// TIA Portal project "test3Servo" (V15.1)

(* hardware
DEVICE "S7-1200 station_1"  S7-1200 Station
   slot 0: "Rack_0"  S7-1200 Rack  Rack  V1.0
   slot 1: "PLC_1"  CPU 1217C DC/DC/DC  6ES7 217-1AG40-0XB0  V4.1
*)

// ===== PLC "PLC_1"  CPU 1217C DC/DC/DC =====

VAR_GLOBAL   // PLC tag table "Default tag table"
   "B1_Pulse" AT %Q0.0 : Bool;
   "B3_Pulse" AT %Q0.2 : Bool;
   "B2_Pulse" AT %Q0.1 : Bool;
   "B3_Direction" AT %Q0.6 : Bool;
   "B2_Direction" AT %Q0.5 : Bool;
   "B1_Direction" AT %Q0.4 : Bool;
   "powerB1" AT %M0.0 : Bool;
   "powerB2" AT %M0.1 : Bool;
   "powerB3" AT %M0.2 : Bool;
   "switch1" AT %I0.0 : Bool;
   "switch2" AT %I0.2 : Bool;
   "switch3" AT %I0.4 : Bool;
   "Tag_1" AT %M4.1 : Bool;
   "Tag_2" AT %MD2 : Real;
END_VAR

DATA_BLOCK "B1"   // DB1, Motion_DB
{ S7_Optimized_Access := 'TRUE' }
AUTHOR : SIMATIC
FAMILY : BasicMC
NAME : TO_PosAx
VERSION : 5.0
// stored: InstanceOfName TO_PositioningAxis
"TO_PositioningAxis"
BEGIN
   // Axis.LengthUnitNormalized.Distance = 1005
   // Axis.DirectionOutputEnabledCU = TRUE
   // Axis.OnlinePtoModeCU = 16#0000_0002
   // Axis.SelectedChannel2EnumCU = %Q0.4
   // Axis.SelectedChannel1EnumCU = %Q0.0
   // Pulse.MinDeltaDeltaFrequencyCU = 0.004
   // Pulse.MaxDeltaDeltaFrequencyCU = 1.0E+10
   // Pulse.MinDeltaFrequencyCU = 0.005
   // Pulse.MaxDeltaFrequencyCU = 9.5E+9
   // Pulse.MinFrequencyCU = 1.0
   // Pulse.MaxFrequencyCU = 1.0E+6
   // Pulse.OutputSourceCU = 16#0000_0000
   // Axis.SelectPTO = 0
   // Axis.LengthUnit.LastDistance = 1005
END_DATA_BLOCK

DATA_BLOCK "B2"   // DB2, Motion_DB
{ S7_Optimized_Access := 'TRUE' }
AUTHOR : SIMATIC
FAMILY : BasicMC
NAME : TO_PosAx
VERSION : 5.0
// stored: InstanceOfName TO_PositioningAxis
"TO_PositioningAxis"
BEGIN
   // Axis.LengthUnitNormalized.Distance = 1005
   // Axis.DirectionOutputEnabledCU = TRUE
   // Axis.OnlinePtoModeCU = 16#0000_0002
   // Axis.SelectedChannel2EnumCU = %Q0.5
   // Axis.SelectedChannel1EnumCU = %Q0.1
   // Pulse.MinDeltaDeltaFrequencyCU = 0.004
   // Pulse.MaxDeltaDeltaFrequencyCU = 1.0E+10
   // Pulse.MinDeltaFrequencyCU = 0.005
   // Pulse.MaxDeltaFrequencyCU = 9.5E+9
   // Pulse.MinFrequencyCU = 1.0
   // Pulse.MaxFrequencyCU = 1.0E+6
   // Pulse.OutputSourceCU = 16#0000_0000
   // Axis.SelectPTO = 1
   // Axis.OnlinePtoIndexCU = 1
   // Axis.LengthUnit.LastDistance = 1005
END_DATA_BLOCK

DATA_BLOCK "B3"   // DB3, Motion_DB
{ S7_Optimized_Access := 'TRUE' }
AUTHOR : SIMATIC
FAMILY : BasicMC
NAME : TO_PosAx
VERSION : 5.0
// stored: InstanceOfName TO_PositioningAxis
"TO_PositioningAxis"
BEGIN
   // Axis.LengthUnitNormalized.Distance = 1005
   // Axis.DirectionOutputEnabledCU = TRUE
   // Axis.OnlinePtoModeCU = 16#0000_0002
   // Axis.SelectedChannel2EnumCU = %Q0.6
   // Axis.SelectedChannel1EnumCU = %Q0.2
   // Pulse.MinDeltaDeltaFrequencyCU = 0.004
   // Pulse.MaxDeltaDeltaFrequencyCU = 1.0E+10
   // Pulse.MinDeltaFrequencyCU = 0.005
   // Pulse.MaxDeltaFrequencyCU = 9.5E+9
   // Pulse.MinFrequencyCU = 1.0
   // Pulse.MaxFrequencyCU = 1.0E+6
   // Pulse.OutputSourceCU = 16#0000_0000
   // Axis.SelectPTO = 2
   // Axis.OnlinePtoIndexCU = 2
   // Axis.LengthUnit.LastDistance = 1005
END_DATA_BLOCK

ORGANIZATION_BLOCK "Main"   // OB1, LAD, ProgramCycle
TITLE = "Main Program Sweep (Cycle)"
{ S7_Optimized_Access := 'TRUE' }
VERSION : 0.1
   VAR_INPUT
      Initial_Call : Bool;   // Initial call of this OB
      Remanence : Bool;   // =True, if remanent data are available
   END_VAR
BEGIN

REGION Network 1
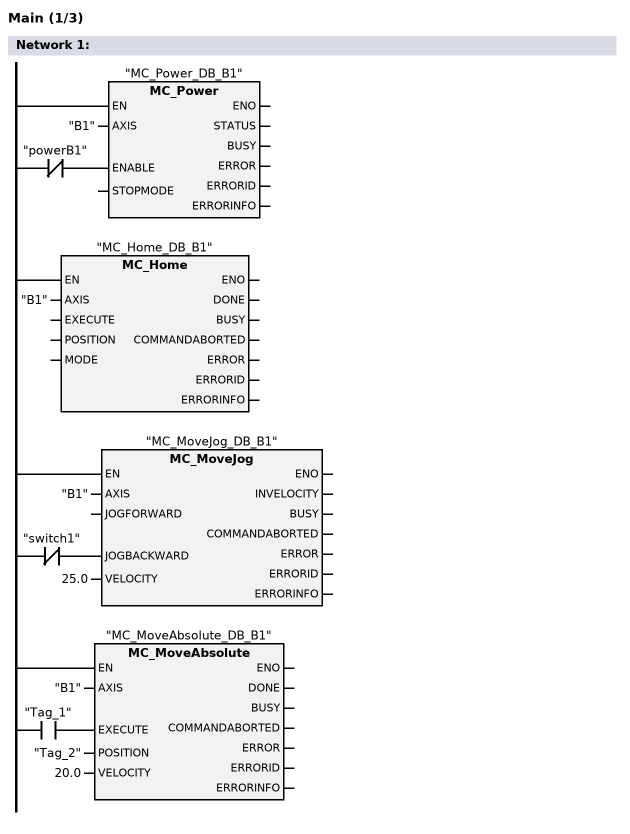
   "MC_Power_DB_B1"(Axis := "B1", Enable := NOT "powerB1");   // MC_Power
   "MC_Home_DB_B1"(Axis := "B1");   // MC_Home
   "MC_MoveJog_DB_B1"(Axis := "B1", JogBackward := NOT "switch1", Velocity := 25.0);   // MC_MoveJog
   "MC_MoveAbsolute_DB_B1"(Axis := "B1", Execute := "Tag_1", Position := "Tag_2", Velocity := 20.0);   // MC_MoveAbsolute
END_REGION

REGION Network 2
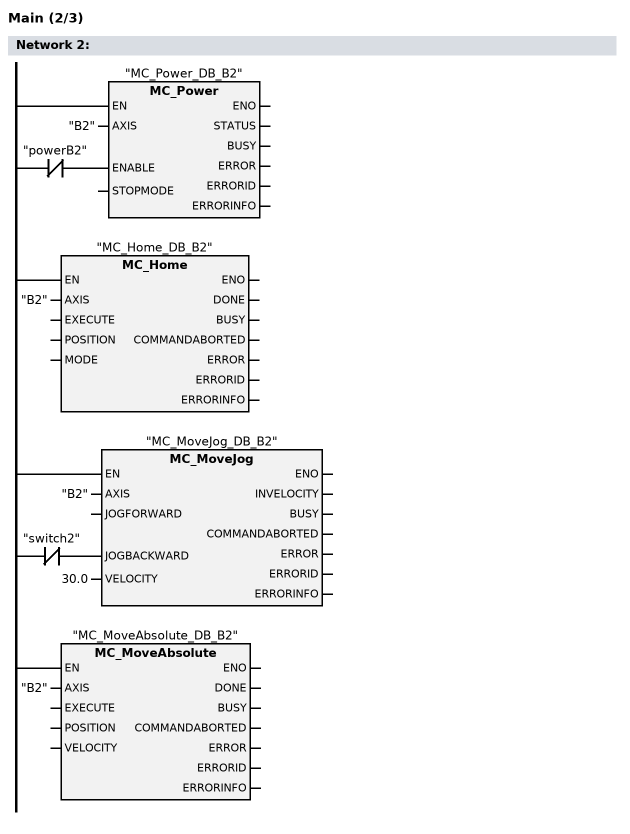
   "MC_Power_DB_B2"(Axis := "B2", Enable := NOT "powerB2");   // MC_Power
   "MC_Home_DB_B2"(Axis := "B2");   // MC_Home
   "MC_MoveJog_DB_B2"(Axis := "B2", JogBackward := NOT "switch2", Velocity := 30.0);   // MC_MoveJog
   "MC_MoveAbsolute_DB_B2"(Axis := "B2");   // MC_MoveAbsolute
END_REGION

REGION Network 3
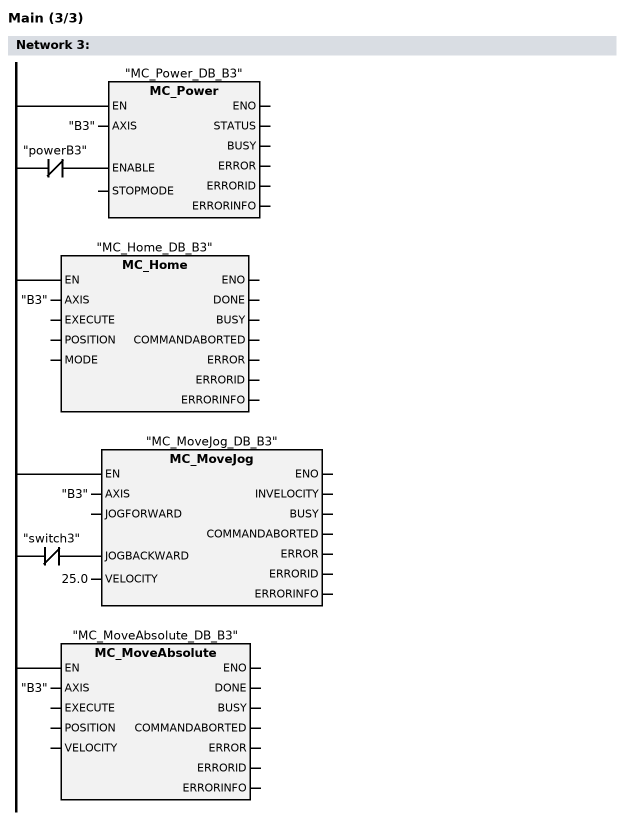
   "MC_Power_DB_B3"(Axis := "B3", Enable := NOT "powerB3");   // MC_Power
   "MC_Home_DB_B3"(Axis := "B3");   // MC_Home
   "MC_MoveJog_DB_B3"(Axis := "B3", JogBackward := NOT "switch3", Velocity := 25.0);   // MC_MoveJog
   "MC_MoveAbsolute_DB_B3"(Axis := "B3");   // MC_MoveAbsolute
END_REGION
END_ORGANIZATION_BLOCK